FUNCTION_BLOCK FB_System_MVHW_Ablaufsteuerung
VAR_IN_OUT
	Zustand					: ST_System_MVHW_Zustand;
	Stellwert				: ST_System_MVHW_Stellwert;
	Steuerung				: ST_System_MVHW_Steuerung;
END_VAR
VAR_INPUT
	Zustand_Stellventil		: ST_SV_Zustand;
	Zustand_Pumpe			: ST_PU_Zustand;
END_VAR
VAR_OUTPUT
END_VAR
VAR
	E_System_DLK_Zustand_Status_Nachl_Stellventil	: SINT;
	E_System_DLK_Zustand_Status_Nachl_Pumpe	: SINT;
	E_System_DLK_Zustand_Status_Betrieb			: SINT;
	E_System_DLK_Zustand_Status_Betrieb_Sperre	: SINT;
	E_System_DLK_Zustand_Status_Vorl_Pumpe		: SINT;
	E_System_DLK_Zustand_Status_Vorl_Stellventil	: SINT;
	E_System_DLK_Zustand_Status_Betriebsbereit	: SINT;
	E_System_DLK_Zustand_Status_Stoerung		: SINT;
	E_System_DLK_Zustand_Status_Idle_Sperre		: SINT;

END_VAR

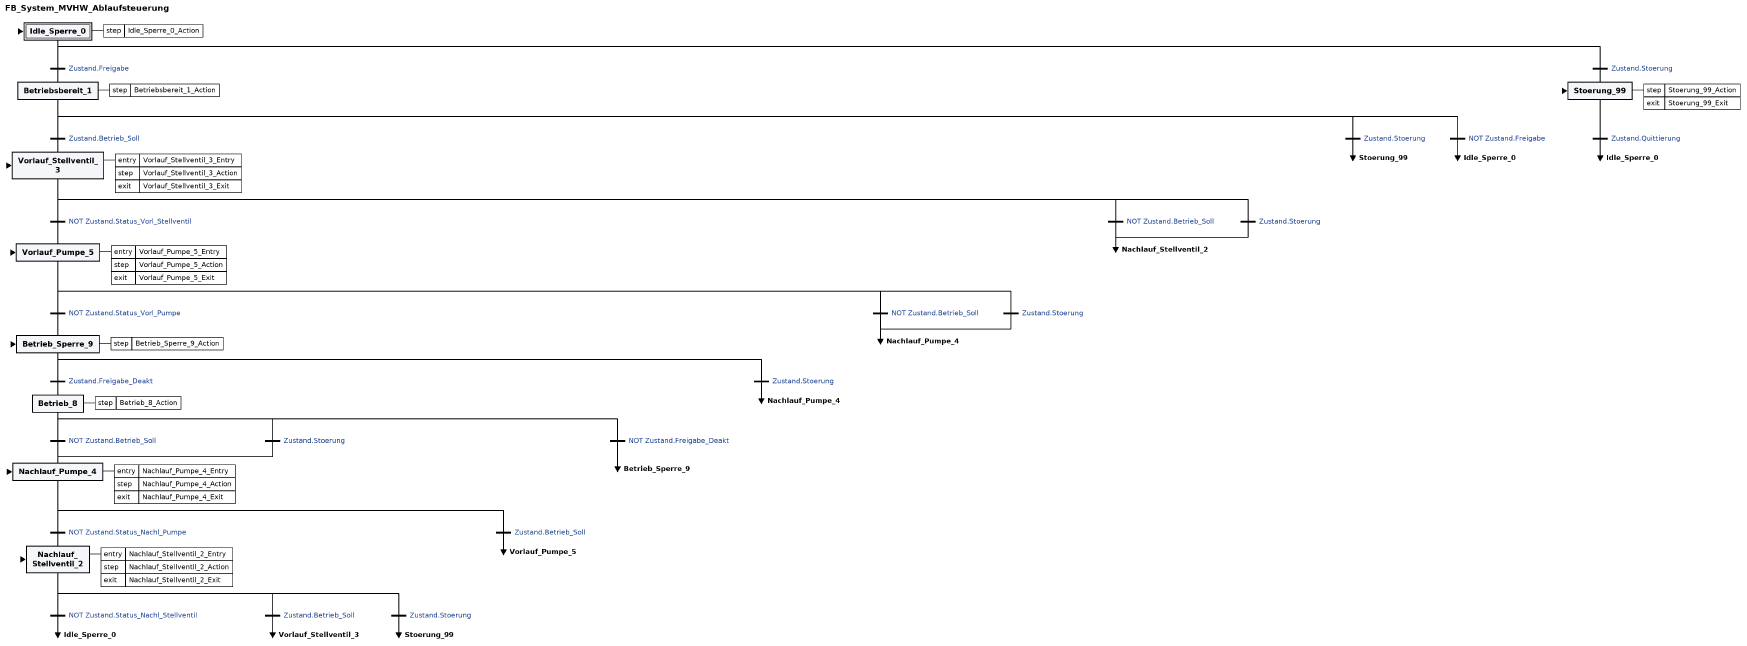
INITIAL_STEP Idle_Sperre_0:
    Idle_Sperre_0_Action(N);  // step action
END_STEP
TRANSITION FROM Idle_Sperre_0 TO Betriebsbereit_1
    := Zustand.Freigabe;
END_TRANSITION
TRANSITION FROM Idle_Sperre_0 TO Stoerung_99
    := Zustand.Stoerung;
END_TRANSITION
STEP Stoerung_99:
    Stoerung_99_Action(N);  // step action
    Stoerung_99_Exit(P0);  // exit action
END_STEP
TRANSITION FROM Stoerung_99 TO Idle_Sperre_0
    := Zustand.Quittierung;
END_TRANSITION
STEP Betriebsbereit_1:
    Betriebsbereit_1_Action(N);  // step action
END_STEP
TRANSITION FROM Betriebsbereit_1 TO Vorlauf_Stellventil_3
    := Zustand.Betrieb_Soll;
END_TRANSITION
TRANSITION FROM Betriebsbereit_1 TO Stoerung_99
    := Zustand.Stoerung;
END_TRANSITION
TRANSITION FROM Betriebsbereit_1 TO Idle_Sperre_0
    := NOT Zustand.Freigabe;
END_TRANSITION
STEP Vorlauf_Stellventil_3:
    Vorlauf_Stellventil_3_Entry(P1);  // entry action
    Vorlauf_Stellventil_3_Action(N);  // step action
    Vorlauf_Stellventil_3_Exit(P0);  // exit action
END_STEP
TRANSITION FROM Vorlauf_Stellventil_3 TO Vorlauf_Pumpe_5
    := NOT Zustand.Status_Vorl_Stellventil;
END_TRANSITION
TRANSITION FROM Vorlauf_Stellventil_3 TO Nachlauf_Stellventil_2
    := NOT Zustand.Betrieb_Soll;
END_TRANSITION
TRANSITION FROM Vorlauf_Stellventil_3 TO Nachlauf_Stellventil_2
    := Zustand.Stoerung;
END_TRANSITION
STEP Vorlauf_Pumpe_5:
    Vorlauf_Pumpe_5_Entry(P1);  // entry action
    Vorlauf_Pumpe_5_Action(N);  // step action
    Vorlauf_Pumpe_5_Exit(P0);  // exit action
END_STEP
TRANSITION FROM Vorlauf_Pumpe_5 TO Betrieb_Sperre_9
    := NOT Zustand.Status_Vorl_Pumpe;
END_TRANSITION
TRANSITION FROM Vorlauf_Pumpe_5 TO Nachlauf_Pumpe_4
    := NOT Zustand.Betrieb_Soll;
END_TRANSITION
TRANSITION FROM Vorlauf_Pumpe_5 TO Nachlauf_Pumpe_4
    := Zustand.Stoerung;
END_TRANSITION
STEP Betrieb_Sperre_9:
    Betrieb_Sperre_9_Action(N);  // step action
END_STEP
TRANSITION FROM Betrieb_Sperre_9 TO Betrieb_8
    := Zustand.Freigabe_Deakt;
END_TRANSITION
TRANSITION FROM Betrieb_Sperre_9 TO Nachlauf_Pumpe_4
    := Zustand.Stoerung;
END_TRANSITION
STEP Betrieb_8:
    Betrieb_8_Action(N);  // step action
END_STEP
TRANSITION FROM Betrieb_8 TO Nachlauf_Pumpe_4
    := NOT Zustand.Betrieb_Soll;
END_TRANSITION
TRANSITION FROM Betrieb_8 TO Nachlauf_Pumpe_4
    := Zustand.Stoerung;
END_TRANSITION
TRANSITION FROM Betrieb_8 TO Betrieb_Sperre_9
    := NOT Zustand.Freigabe_Deakt;
END_TRANSITION
STEP Nachlauf_Pumpe_4:
    Nachlauf_Pumpe_4_Entry(P1);  // entry action
    Nachlauf_Pumpe_4_Action(N);  // step action
    Nachlauf_Pumpe_4_Exit(P0);  // exit action
END_STEP
TRANSITION FROM Nachlauf_Pumpe_4 TO Nachlauf_Stellventil_2
    := NOT Zustand.Status_Nachl_Pumpe;
END_TRANSITION
TRANSITION FROM Nachlauf_Pumpe_4 TO Vorlauf_Pumpe_5
    := Zustand.Betrieb_Soll;
END_TRANSITION
STEP Nachlauf_Stellventil_2:
    Nachlauf_Stellventil_2_Entry(P1);  // entry action
    Nachlauf_Stellventil_2_Action(N);  // step action
    Nachlauf_Stellventil_2_Exit(P0);  // exit action
END_STEP
TRANSITION FROM Nachlauf_Stellventil_2 TO Idle_Sperre_0
    := NOT Zustand.Status_Nachl_Stellventil;
END_TRANSITION
TRANSITION FROM Nachlauf_Stellventil_2 TO Vorlauf_Stellventil_3
    := Zustand.Betrieb_Soll;
END_TRANSITION
TRANSITION FROM Nachlauf_Stellventil_2 TO Stoerung_99
    := Zustand.Stoerung;
END_TRANSITION

ACTION Betrieb_8_Action:
(* Stellwert setzen *)
Stellwert.Anford_Stellventil		:= TRUE;
Stellwert.Anford_Pumpe		:= TRUE;
Stellwert.Anford_Kompressor			:= TRUE;

(* Zustand setzen *)
Zustand.Status				:= E_System_DLK_Zustand_Status_Betrieb;
END_ACTION

ACTION Betrieb_Sperre_9_Action:
(* Stellwert setzen *)
Stellwert.Anford_Stellventil		:= TRUE;
Stellwert.Anford_Pumpe		:= TRUE;
Stellwert.Anford_Kompressor			:= TRUE;

(* Zustand setzen *)
Zustand.Status				:= E_System_DLK_Zustand_Status_Betrieb_Sperre;
END_ACTION

ACTION Betriebsbereit_1_Action:
(* Stellwert setzen *)
Stellwert.Anford_Stellventil	:= FALSE;
Stellwert.Anford_Pumpe	:= FALSE;
Stellwert.Anford_Kompressor		:= FALSE;

(* Zustand setzen *)
Zustand.Status			:= E_System_DLK_Zustand_Status_Betriebsbereit;
END_ACTION

ACTION Idle_Sperre_0_Action:
(* Stellwert setzen *)
Stellwert.Anford_Stellventil	:= FALSE;
Stellwert.Anford_Pumpe	:= FALSE;
Stellwert.Anford_Kompressor		:= FALSE;

(* Zustand setzen *)
Zustand.Status			:= E_System_DLK_Zustand_Status_Idle_Sperre;

(* Quittierungszustand auf False setzen, damit das System bei einer erneuten Störung nicht direkt wieder angeschaltet wird *)
Steuerung.Quittierung	:= FALSE;
END_ACTION

ACTION Nachlauf_Pumpe_4_Action:
(* Stellwert setzen *)
Stellwert.Anford_Stellventil		:= TRUE;
Stellwert.Anford_Pumpe		:= FALSE;
Stellwert.Anford_Kompressor			:= FALSE;

(* Zustand setzen *)
Zustand.Status				:= E_System_DLK_Zustand_Status_Nachl_Pumpe;
Zustand.Status_Nachl_Pumpe	:= Zustand_Pumpe.Betrieb OR Zustand_Pumpe.Status_Nachl;
END_ACTION

ACTION Nachlauf_Pumpe_4_Entry:
Zustand.Status_Nachl_Pumpe	:= TRUE;
END_ACTION

ACTION Nachlauf_Pumpe_4_Exit:
Zustand.Status_Nachl_Pumpe	:= FALSE;
END_ACTION

ACTION Nachlauf_Stellventil_2_Action:
(* Stellwert setzen *)
Stellwert.Anford_Stellventil		:= FALSE;
Stellwert.Anford_Pumpe		:= FALSE;
Stellwert.Anford_Kompressor			:= FALSE;

(* Zustand setzen *)
Zustand.Status				:= E_System_DLK_Zustand_Status_Nachl_Stellventil;
Zustand.Status_Nachl_Stellventil	:= Zustand_Stellventil.Stellung OR Zustand_Stellventil.Stellungwechsel10;
END_ACTION

ACTION Nachlauf_Stellventil_2_Entry:
Zustand.Status_Nachl_Stellventil	:= TRUE;
END_ACTION

ACTION Nachlauf_Stellventil_2_Exit:
Zustand.Status_Nachl_Stellventil	:= FALSE;
END_ACTION

ACTION Stoerung_99_Action:
(* Stellwert setzen *)
Stellwert.Anford_Stellventil	:= FALSE;
Stellwert.Anford_Pumpe	:= FALSE;
Stellwert.Anford_Kompressor		:= FALSE;

(* Zustand setzen *)
Zustand.Stoerung			:= TRUE;
Zustand.Status			:= E_System_DLK_Zustand_Status_Stoerung;
END_ACTION

ACTION Stoerung_99_Exit:
Zustand.Stoerung	:= FALSE;
END_ACTION

ACTION Vorlauf_Pumpe_5_Action:
(* Stellwert setzen *)
Stellwert.Anford_Stellventil		:= TRUE;
Stellwert.Anford_Pumpe				:= TRUE;
Stellwert.Anford_Kompressor			:= FALSE;

(* Zustand setzen *)
Zustand.Status				:= E_System_DLK_Zustand_Status_Vorl_Pumpe;
Zustand.Status_Vorl_Pumpe	:= NOT(Zustand_Pumpe.Betrieb AND NOT Zustand_Pumpe.Status_Vorl);
END_ACTION

ACTION Vorlauf_Pumpe_5_Entry:
Zustand.Status_Vorl_Pumpe	:= TRUE;
END_ACTION

ACTION Vorlauf_Pumpe_5_Exit:
Zustand.Status_Vorl_Pumpe	:= FALSE;
END_ACTION

ACTION Vorlauf_Stellventil_3_Action:
(* Stellwert setzen *)
Stellwert.Anford_Stellventil		:= TRUE;
Stellwert.Anford_Pumpe		:= FALSE;
Stellwert.Anford_Kompressor			:= FALSE;

(* Zustand setzen *)
Zustand.Status				:= E_System_DLK_Zustand_Status_Vorl_Stellventil;
Zustand.Status_Vorl_Stellventil	:= NOT(Zustand_Stellventil.Stellung AND NOT Zustand_Stellventil.Stellungwechsel01);
END_ACTION

ACTION Vorlauf_Stellventil_3_Entry:
Zustand.Status_Vorl_Stellventil	:= TRUE;
END_ACTION

ACTION Vorlauf_Stellventil_3_Exit:
Zustand.Status_Vorl_Stellventil	:= FALSE;
END_ACTION

END_FUNCTION_BLOCK

(* stored: Version 1.1.0.1, ProductVersion 3.1.4024.9
   POU FB_System_MVHW_Ablaufsteuerung: Id {f5500d41-5722-44b2-abde-83ffacb69035}, SpecialFunc None
   Action Betrieb_8_Action: Id {b5653d0c-8af9-4b77-aef4-eebecc7eb20a}
   Action Betrieb_Sperre_9_Action: Id {1e31951b-1936-4599-9098-4ede0ee24f3e}
   Action Betriebsbereit_1_Action: Id {67400e1d-8caf-46fb-8cac-dcc9bf8ad325}
   Action Idle_Sperre_0_Action: Id {e9c71f31-5b49-45e6-96f8-11d09f04d7c5}
   Action Nachlauf_Pumpe_4_Action: Id {f42f7ec6-00a8-48aa-93bb-8ef557ca7547}
   Action Nachlauf_Pumpe_4_Entry: Id {243fe88a-ca98-46e3-baf7-930db52b4a19}
   Action Nachlauf_Pumpe_4_Exit: Id {0338e721-f612-4b37-a3f0-607c25b49dca}
   Action Nachlauf_Stellventil_2_Action: Id {aabb0b81-c96d-4aa5-9a81-f4e749c89dd0}
   Action Nachlauf_Stellventil_2_Entry: Id {3600e4a2-803c-4bb7-8fda-6c1fc59c8e60}
   Action Nachlauf_Stellventil_2_Exit: Id {a3a1e283-ee71-4312-94d0-52053ceb2cbb}
   Action Stoerung_99_Action: Id {ad522ac5-34ee-4b32-bf6f-5107997929dc}
   Action Stoerung_99_Exit: Id {bd1614e0-d55f-4fe3-be6b-4f8744077873}
   Action Vorlauf_Pumpe_5_Action: Id {53c608ec-97b3-4251-9929-91c7c4aa931a}
   Action Vorlauf_Pumpe_5_Entry: Id {fca47273-738b-4665-b89f-a25400875b55}
   Action Vorlauf_Pumpe_5_Exit: Id {67b823e4-1003-4422-9102-dc09e123e652}
   Action Vorlauf_Stellventil_3_Action: Id {410dd3fa-429d-4576-ab98-45a37bd49784}
   Action Vorlauf_Stellventil_3_Entry: Id {81853fad-3887-4397-bb94-bbd594aa0df0}
   Action Vorlauf_Stellventil_3_Exit: Id {5e54dac3-83f9-46e1-924b-8753a862e695} *)
